ORGANIZATION_BLOCK MAIN:OB1
TITLE=PROGRAM COMMENTS
BEGIN
Network 1 // Make a Logic when I0.0 is ON, Q0.0 is ON & Q0.1 is OFF & when I0.0 is OFF, Q0.1 should be ON & Q0.0 should be OFF
LD     I0.0
=      Q0.0
Network 2
LDN    Q0.0
=      Q0.1
END_ORGANIZATION_BLOCK
SUBROUTINE_BLOCK SBR_0:SBR0
TITLE=SUBROUTINE COMMENTS
BEGIN
Network 1 // Network Title
// Network Comment
END_SUBROUTINE_BLOCK
INTERRUPT_BLOCK INT_0:INT0
TITLE=INTERRUPT ROUTINE COMMENTS
BEGIN
Network 1 // Network Title
// Network Comment
END_INTERRUPT_BLOCK
